Yaskawa INFORM job: CLEAN-R1_KM.JBI

/JOB
//NAME CLEAN-R1_KM
///FOLDERNAME CLEAN
//POS
///NPOS 21,21,0,0,0,0
///TOOL 0
///POSTYPE PULSE
///PULSE
C00000=3643,-76224,-106676,19950,71810,76872
C00001=2508,0,0,0,0,4169
C00002=41115,93452,-30342,-19926,115521,85678
C00003=28599,109925,-13759,-12658,112881,84157
C00004=28301,105457,-14309,-12299,110948,84323
C00005=28966,99224,-20084,-13542,107459,84155
C00006=29027,99166,-20392,-13590,107618,84144
C00007=28599,108424,-14443,-12622,112541,84195
C00008=34011,109773,-12073,-16636,107751,84808
C00009=32816,112629,-5671,-14598,109695,85231
C00010=32618,110353,-5730,-14378,108579,85337
C00011=32545,109523,-5728,-14298,108158,85375
C00012=32618,110353,-5730,-14378,108579,85337
C00013=32816,112629,-5671,-14598,109695,85231
C00014=34011,109773,-12073,-16636,107751,84808
C00015=38810,111241,-7992,-19438,105697,85727
C00016=36913,114349,813,-16982,106196,86149
C00017=37169,116704,797,-17245,107389,86018
C00018=39968,92120,-23778,-21749,94252,85800
C00019=46315,71110,-54300,-23622,119041,85704
C00020=32571,-80067,-84751,-11816,58952,90735
BC00000=199464,674570,1075173
BC00001=0,0,0
BC00002=204899,578,1075157
BC00003=204899,578,1075157
BC00004=204899,578,1075157
BC00005=204899,578,1075157
BC00006=204899,578,1075157
BC00007=204899,578,1075157
BC00008=204899,578,1075157
BC00009=204899,578,1075157
BC00010=204899,578,1075157
BC00011=204899,578,1075157
BC00012=204899,578,1075157
BC00013=204899,578,1075157
BC00014=204899,578,1075157
BC00015=204899,578,1075157
BC00016=204894,578,1075156
BC00017=204894,578,1075156
BC00018=204894,578,1075156
BC00019=204899,578,1075157
BC00020=204899,578,820586
//INST
///DATE 2024/02/27 11:42
///ATTR SC,RW
///GROUP1 RB1,BS1
///LVARS 0,5,0,0,0,3,3,0
NOP
MOVJ C00000 BC00000 VJ=100.00
SFTOF
'********************************
'Please check position before
'running in play-mode
'********************************
'#Output - Cleaning Motor
SET LI000 14
'#Output - Cleaning Oil
SET LI001 15
'#Output - Wirecut
SET LI002 16
'#Output - Wirefeeder Forward
SET LI003 4095
'#Output - Torch Blow out
SET LI004 4091
'********************************
REFP 1 C00001 BC00001
GETS LPX001 $PX011
CNVRT LPX001 LPX001 RF
GETS LPX002 $PX001
CNVRT LPX002 LPX002 RF
SUB LBP002 LBP001
'Comment out axis to shift
SETE LBP002 (1) 0
COMM SETE LBP002 (2) 0
SETE LBP002 (3) 0
SFTON LBP002
'********************************
'SAFE POS
PAUSE IF IN#(1563)=OFF
MOVJ C00002 BC00002 VJ=100.00
'WIRECUT
MOVJ C00003 BC00003 VJ=100.00
'WIREFEED OUTPUT
PULSE OT#(LI003) T=0.80
MOVL C00004 BC00004 V=133.3
MOVL C00005 BC00005 V=66.7
TIMER T=0.20
DOUT OT#(LI002) ON
TIMER T=1.00
MOVL C00006 BC00006 V=166.7
MOVL C00007 BC00007 V=333.3
DOUT OT#(LI002) OFF
'CLEANING MOTOR
MOVJ C00008 BC00008 VJ=50.00
MOVL C00009 BC00009 V=250.0
'CLEANING AIR
DOUT OT#(LI004) ON
MOVL C00010 BC00010 V=50.0
TIMER T=0.20
DOUT OT#(LI000) ON
TIMER T=0.50
MOVL C00011 BC00011 V=25.0
TIMER T=0.50
MOVL C00012 BC00012 V=25.0
TIMER T=0.20
DOUT OT#(LI000) OFF
TIMER T=0.50
DOUT OT#(LI004) OFF
MOVL C00013 BC00013 V=25.0
MOVL C00014 BC00014 V=333.3
'CLEANING OIL
MOVJ C00015 BC00015 VJ=50.00
MOVL C00016 BC00016 V=100.0
PULSE OT#(LI001) T=0.20
TIMER T=1.00
MOVL C00017 BC00017 V=333.3
'CLEANING AIR
PULSE OT#(LI004) T=1.00
TIMER T=1.00
MOVJ C00018 BC00018 VJ=40.00
'SAFE POS
MOVJ C00019 BC00019 VJ=100.00
MOVJ C00020 BC00020 VJ=100.00
SFTOF
'********************************
'*         CLEANING JOB         *
'*      __ __ _____ _____       *
'*     |  |  |   | | __  |      *
'*     |_   _| | | |    -|      *
'*       |_| |_|___|__|__|      *
'*        YRC Multi Base        *
'*       rev 4. 2021-10-12      *
'********************************
END
